// TIA Portal V20 export
TYPE "LBP_typeModularMcpModeGroupOutput"
TITLE = Modular MCP image / Image MCP modulaire
// Output image of mode group keypad for modular MCP / Image des sorties du pupitre de groupes de modes de fonctionnement pour MCP modulaires
   STRUCT
      reset : Bool;   // output image n+0 bit 0 / Image des sorties n+0 bit 0
      cycleStop : Bool;   // output image n+0 bit 1 / Image des sorties n+0 bit 1
      cycleStart : Bool;   // output image n+0 bit 2 / Image des sorties n+0 bit 2
      singleBlock : Bool;   // output image n+0 bit 3 / Image des sorties n+0 bit 3
      inc100 : Bool;   // output image n+0 bit 4 / Image des sorties n+0 bit 4
      inc1000 : Bool;   // output image n+0 bit 5 / Image des sorties n+0 bit 5
      auto : Bool;   // output image n+0 bit 6 / Image des sorties n+0 bit 6
      inc1 : Bool;   // output image n+0 bit 7 / Image des sorties n+0 bit 7
      inc10 : Bool;   // output image n+1 bit 0 / Image des sorties n+1 bit 0
      mda : Bool;   // output image n+1 bit 1 / Image des sorties n+1 bit 1
      teachIn : Bool;   // output image n+1 bit 2 / Image des sorties n+1 bit 2
      incVar : Bool;   // output image n+1 bit 3 / Image des sorties n+1 bit 3
      jog : Bool;   // output image n+1 bit 4 / Image des sorties n+1 bit 4
      repos : Bool;   // output image n+1 bit 5 / Image des sorties n+1 bit 5
      refPoint : Bool;   // output image n+1 bit 6 / Image des sorties n+1 bit 6
      reserved17 : Bool;
      led16 : Bool;   // output image n+2 bit 0 / Image des sorties n+2 bit 0
      led17 : Bool;   // output image n+2 bit 1 / Image des sorties n+2 bit 1
      led18 : Bool;   // output image n+2 bit 2 / Image des sorties n+2 bit 2
      reserved23 : Bool;
      reserved24 : Bool;
      reserved25 : Bool;
      reserved26 : Bool;
      reserved27 : Bool;
      led24 : Bool;   // output image n+3 bit 0 / Image des sorties n+3 bit 0
      led25 : Bool;   // output image n+3 bit 1 / Image des sorties n+3 bit 1
      led26 : Bool;   // output image n+3 bit 2 / Image des sorties n+3 bit 2
      reserved33 : Bool;
      reserved34 : Bool;
      reserved35 : Bool;
      reserved36 : Bool;
      reserved37 : Bool;
   END_STRUCT;
END_TYPE
